{attribute addProperty ShortName ""}
FUNCTION_BLOCK ABSTRACT CUBase EXTENDS TcoCore.TcoObject IMPLEMENTS ICUBase

VAR
    _cuId        : eStations;
    _processData : ProcessDataManager(THIS^);
	_groupInspection : TcoInspectors.TcoInspectionGroup(THIS^);
	{attribute addProperty Name "<#STATUS INFO#>"}
    _statusInfo  : CUBaseStatusInfo := (Parent := THIS^);
	_operatorInfo : OperatorInfo := (Parent := THIS^);
	_settings  : CUBaseSettings := (Parent := THIS^);
	//~
	_toggle: TcoUtilities.TcoBlinker(THIS^);
	//~
	_recurringFails:CuBaseRecurringFailures:=(Parent:=THIS^);
	_productionPlaner:ProductionPlaner(THIS^);
	_internalData : REFERENCE TO InternalStorage;	
	
	{attribute clr [ReadOnly()]}
	{attribute clr [RenderIgnore()]}
	_readyForOperations : BOOL;
END_VAR

(*~
	<docu>
		<summary>
			Controls `automatic` mode of `CU00x`.
		</summary>
	</docu>
~*)
METHOD  Automat
VAR_INPUT
END_VAR
(*
	Enable condition to start `automatTask`.
	Modify according your needs.
	[! 
	THIS IS NOT SAFETY CONDITION. THE SAFETY OF PRESONNEL AND EQUIPMENT MUST BE ENSURED BY ADDITIONAL MEANS 
	TO COMPLY WITH REGULATIONS
	]
*)


AutomatTask.Task.Enabled :=  AutomatTask.Task.Busy  XOR
							(GroundTask.GroundDone AND NOT AutomatTask.Task.Busy AND THIS^.Technology.AllowAutomat(inCuId:=CuId));

(*
	Invokes `groundTask` from technology object.
*)

IF(Technology.AutomatAllTask.Execute()) THEN AutomatTask.Task.Invoke(); END_IF;

IF(Technology.ForceStepMode()) THEN
 	AutomatTask.ModeController.Mode := eSequencerMode.StepMode;
END_IF
END_METHOD

PROPERTY ABSTRACT AutomatTask : REFERENCE TO CUBaseAutomat
GET
END_GET
END_PROPERTY

PROPERTY  CreateEntityTask : TcoCore.ITcoTaskStatus
GET
CreateEntityTask := _processData._createTask;
END_GET
END_PROPERTY

PROPERTY CuId : eStations
GET
CuId := _cuId;
END_GET
SET
_cuId := CuId;
END_SET
END_PROPERTY

PROPERTY  DeleteEntityTask : TcoCore.ITcoTaskStatus
GET
DeleteEntityTask := _processData._deleteTask;
END_GET
END_PROPERTY

METHOD DoesBelong : BOOL
DoesBelong := THIS^.ProcessDataManager.Data.EntityHeader.NextStation = THIS^.CuId;
END_METHOD

METHOD EntityFlowCloseForOperations : TcoCore.ITcoTaskStatus
VAR_IN_OUT
	Header : CuHeader; 
END_VAR
THIS^.FlagCloseEntity(Header);
EntityFlowCloseForOperations := THIS^.ProcessDataManager.Update(ProcessDataManager.Data._EntityId);
END_METHOD

METHOD EntityFlowCreateNew : TcoCore.ITcoTaskStatus
VAR_INPUT
	EntityId : STRING(255);	
END_VAR
VAR_IN_OUT
	Header : CuHeader;
END_VAR
THIS^.FlagCreateNewEntity(EntityId, Header);
EntityFlowCreateNew := THIS^.ProcessDataManager.Create(EntityId);
END_METHOD

METHOD EntityFlowDiscard : TcoCore.ITcoTaskStatus
VAR_INPUT
	EntityId : STRING(255);	
END_VAR
VAR_IN_OUT	
	Header : CuHeader; 
END_VAR
THIS^.FlagThrowAwayEntity(Header);
EntityFlowDiscard := THIS^.ProcessDataManager.Update(EntityId);
END_METHOD

METHOD EntityFlowFinalize : TcoCore.ITcoTaskStatus
VAR_IN_OUT
	Header : CuHeader; 
END_VAR
THIS^.FlagFinishEntity(Header);
EntityFlowFinalize := THIS^.ProcessDataManager.Update(ProcessDataManager.Data._EntityId);
END_METHOD

METHOD EntityFlowOpenForOperations : TcoCore.ITcoTaskStatus
VAR_INPUT
	Identifier : STRING(255);	
END_VAR
VAR_IN_OUT
	Header : CuHeader;
END_VAR
EntityFlowOpenForOperations := THIS^.ProcessDataManager.Read(Identifier);
THIS^.FlagOpenEntity(Identifier, Header);
END_METHOD

PROPERTY  ExistEntityTask : TcoCore.ITcoTaskStatus
GET
ExistEntityTask := _processData._idExistsTask;
END_GET
END_PROPERTY

METHOD PRIVATE FlagCloseEntity : BOOL
VAR_IN_OUT
	Header : CuHeader; 
END_VAR
THIS^.ProcessDataManager.Data.EntityHeader.LastStation := THIS^.CuId;

IF(THIS^.ProcessDataManager.Data.EntityHeader.Results.Result = TcoInspectors.eOverallResult.Failed) THEN	
	THIS^.ProcessDataManager.Data.EntityHeader.NextStation := Header.NextOnFailed;
ELSIF(THIS^.ProcessDataManager.Data.EntityHeader.Results.Result = TcoInspectors.eOverallResult.Passed) THEN
	THIS^.ProcessDataManager.Data.EntityHeader.NextStation := Header.NextOnPassed;
ELSIF(THIS^.ProcessDataManager.Data.EntityHeader.Results.Result = TcoInspectors.eOverallResult.InProgress) THEN
	THIS^.ProcessDataManager.Data.EntityHeader.NextStation := Header.NextOnPassed;
END_IF

THIS^.ProcessDataManager.Data.EntityHeader.OpenOn := eStations.NONE;
Header.CycleTime := THIS^._statusInfo.CurrentCycleTime;
Header.CleanLoopTime := THIS^._statusInfo.CurrentCleanCycleTime;
Header.OperationsEnded := Context.RealTimeClock.NowLocal();
Header.Operator := _operatorInfo.UserName;
END_METHOD

METHOD PRIVATE FlagCreateNewEntity : BOOL
VAR_INPUT
	Identifier : STRING(255);	
END_VAR
VAR_IN_OUT
	Header : CuHeader;
END_VAR
THIS^.ProcessDataManager.Data.EntityHeader.Results.Result := TcoInspectors.eOverallResult.InProgress;
THIS^.ProcessDataManager.Data._EntityId := Identifier;
THIS^.ProcessDataManager.Data.EntityHeader.WasReset := FALSE;
END_METHOD

METHOD PRIVATE FlagFinishEntity : BOOL
VAR_IN_OUT
	Header : CuHeader; 
END_VAR
THIS^.ProcessDataManager.Data.EntityHeader.LastStation := THIS^.CuId;

IF(THIS^.ProcessDataManager.Data.EntityHeader.Results.Result = TcoInspectors.eOverallResult.InProgress) THEN
	THIS^.ProcessDataManager.Data.EntityHeader.Results.Result := TcoInspectors.eOverallResult.Passed;
END_IF

IF(THIS^.ProcessDataManager.Data.EntityHeader.Results.Result = TcoInspectors.eOverallResult.Failed) THEN	
	THIS^.ProcessDataManager.Data.EntityHeader.NextStation := Header.NextOnFailed;
ELSIF(THIS^.ProcessDataManager.Data.EntityHeader.Results.Result = TcoInspectors.eOverallResult.Passed) THEN
	THIS^.ProcessDataManager.Data.EntityHeader.NextStation := Header.NextOnPassed;
END_IF

THIS^.ProcessDataManager.Data.EntityHeader.OpenOn := eStations.NONE;

Header.CycleTime := THIS^._statusInfo.CurrentCycleTime;
Header.CleanLoopTime := THIS^._statusInfo.CurrentCleanCycleTime;
Header.OperationsEnded := Context.RealTimeClock.NowLocal();
Header.Operator := _operatorInfo.UserName;
END_METHOD

METHOD PRIVATE FlagOpenEntity : BOOL
VAR_INPUT
	Identifier : STRING(255);	
END_VAR
VAR_IN_OUT
	Header : CuHeader;
END_VAR
Header.Operator := _operatorInfo.UserName;
Header.OperationsStarted := Context.RealTimeClock.NowLocal();
THIS^.ProcessDataManager.Data.EntityHeader.Results.Result := TcoInspectors.eOverallResult.InProgress;
THIS^.ProcessDataManager.Data._EntityId := Identifier;
THIS^.ProcessDataManager.Data.EntityHeader.OpenOn := THIS^.CuId;
THIS^.ProcessDataManager.Data.EntityHeader.WasReset := FALSE;
END_METHOD

METHOD PRIVATE FlagThrowAwayEntity : BOOL
VAR_IN_OUT	
	CuHeader : CuHeader; 
END_VAR
IF(THIS^.ProcessDataManager.Data.EntityHeader.OpenOn <> eStations.NONE) THEN
	THIS^.ProcessDataManager.Data.EntityHeader.LastStation := THIS^.CuId;
	THIS^.ProcessDataManager.Data.EntityHeader.NextStation := CuHeader.NextOnFailed;
	THIS^.ProcessDataManager.Data.EntityHeader.Results.Result := TcoInspectors.eOverallResult.Failed;
	THIS^.ProcessDataManager.Data.EntityHeader.WasReset := TRUE;
END_IF;
END_METHOD

(*~
	<docu>
		<summary>
			Controls `ground` mode of `CU00x`.
		</summary>
	</docu>
~*)
METHOD Ground : BOOL
VAR_INPUT
END_VAR
(*
	Enable condition to start `groundTask`.
	Modify according your needs.
	[! 
	THIS IS NOT SAFETY CONDITION. THE SAFETY OF PRESONNEL AND EQUIPMENT MUST BE ENSURED BY ADDITIONAL MEANS 
	TO COMPLY WITH REGULATIONS
	]
*)

GroundTask.Task.Enabled :=  THIS^.Technology.AllowGround(inCuId:=CuId)  OR GroundTask.Task.Busy ;

(*
	Invokes `groundTask` from technology object.
*)


IF(Technology.GroundAllTask.Execute()) THEN GroundTask.Restore();GroundTask.Task.Invoke(); END_IF;


IF GroundTask.GroundDone AND GroundTask.Task.Execute() THEN GroundTask.Restore();GroundTask.Task.Invoke();END_IF;
END_METHOD

PROPERTY ABSTRACT GroundTask : REFERENCE TO CUBaseGround
GET
END_GET
END_PROPERTY

PROPERTY FINAL GroupInspection : REFERENCE TO TcoInspectionGroup
GET
GroupInspection REF= _groupInspection;
END_GET
END_PROPERTY

(*~
	<docu>
		<summary>
			Code to be called cylically when `CU00x` idle; no other mode is active.
		</summary>
	</docu>
~*)
METHOD Idle : BOOL
END_METHOD

METHOD InternalCloseEntity : BOOL
VAR_INPUT
	inCarrier : UINT;
	refStorage : REFERENCE TO InternalStorage;
END_VAR
VAR_IN_OUT
	inoHeader : CuHeader; 
END_VAR
VAR_INST
	_internalData : REFERENCE TO InternalStorage;	
END_VAR
THIS^.FlagCloseEntity(inoHeader);
_internalData REF= refStorage;
InternalCloseEntity := _internalData.SaveByCarrier(inCarrier, THIS^.ProcessDataManager.Data);
END_METHOD

METHOD InternalCreateNewEntity : BOOL
VAR_INPUT
	inCarrier : UINT;
	refStorage : REFERENCE TO InternalStorage;
END_VAR
VAR_IN_OUT
	inoHeader : CuHeader; 
END_VAR
VAR_INST
	_internalData : REFERENCE TO InternalStorage;	
END_VAR
THIS^.FlagCreateNewEntity(UINT_TO_STRING(inCarrier), inoHeader);
THIS^.ProcessDataManager.Data.EntityHeader.Carrier := UINT_TO_STRING(inCarrier);
_internalData REF= refStorage;
InternalCreateNewEntity := _internalData.SaveByCarrier(inCarrier, THIS^.ProcessDataManager.Data);
END_METHOD

METHOD InternalFinishEntity : BOOL
VAR_INPUT
	inCarrier : UINT;
	refStorage : REFERENCE TO InternalStorage;
END_VAR
VAR_IN_OUT
	inoHeader : CuHeader; 
END_VAR
VAR_INST
	_internalData : REFERENCE TO InternalStorage;	
END_VAR
THIS^.FlagFinishEntity(inoHeader);

_internalData REF= refStorage;
InternalFinishEntity := _internalData.SaveByCarrier(inCarrier, THIS^.ProcessDataManager.Data);
END_METHOD

METHOD InternalOpenEntity : BOOL
VAR_INPUT
	inCarrier : UINT;
	refStorage : REFERENCE TO InternalStorage;
END_VAR
VAR_IN_OUT
	inoHeader : CuHeader; 
END_VAR
VAR_INST
	_internalData : REFERENCE TO InternalStorage;	
END_VAR
_internalData REF= refStorage;
InternalOpenEntity := _internalData.GetByCarrier(inCarrier, THIS^.ProcessDataManager.Data);
THIS^.FlagOpenEntity(UINT_TO_STRING(inCarrier), inoHeader);
END_METHOD

METHOD InternalRetrieveEntity : BOOL
VAR_INPUT
	inCarrier : UINT;
	refStorage : REFERENCE TO InternalStorage;
END_VAR
VAR_INST
	_internalData : REFERENCE TO InternalStorage;	
END_VAR
_internalData REF= refStorage;
InternalRetrieveEntity := _internalData.GetByCarrier(inCarrier, THIS^.ProcessDataManager.Data);
END_METHOD

METHOD InternalThrowAwayEntity : BOOL
VAR_INPUT
	inCarrier : UINT;
	refStorage : REFERENCE TO InternalStorage;
END_VAR
VAR_IN_OUT
	inoHeader : CuHeader; 
END_VAR
VAR_INST
	_internalData : REFERENCE TO InternalStorage;	
END_VAR
THIS^.FlagThrowAwayEntity(inoHeader);
_internalData REF= refStorage;
InternalThrowAwayEntity := _internalData.SaveByCarrier(inCarrier, THIS^.ProcessDataManager.Data);
END_METHOD

(*~
	<docu>
		<summary>
			Controls `manual` mode of `CU00x`.
		</summary>
	</docu>
~*)
METHOD Manual : BOOL
VAR_INPUT
END_VAR
(*
	Enable condition to start `automatTask`.
	Modify according your needs.
	[! 
	THIS IS NOT SAFETY CONDITION. THE SAFETY OF PRESONNEL AND EQUIPMENT MUST BE ENSURED BY ADDITIONAL MEANS 
	TO COMPLY WITH REGULATIONS
	]
*)

ManualTask.Task.Enabled :=  THIS^.Technology.AllowManual(inCuId:=CuId)  OR ManualTask.Task.Busy;
END_METHOD

PROPERTY ABSTRACT ManualTask : REFERENCE TO TcoTaskedService
GET
END_GET
END_PROPERTY

PROPERTY FINAL ProcessDataManager : REFERENCE TO ProcessDataManager
GET
ProcessDataManager REF= _processData;
END_GET
END_PROPERTY

PROPERTY  ReadEntityTask : TcoCore.ITcoTaskStatus
GET
ReadEntityTask := _processData._readTask;
END_GET
END_PROPERTY

METHOD ReadyForOperations : BOOL
VAR_INPUT
END_VAR
ReadyForOperations := _readyForOperations;
END_METHOD

PROPERTY ABSTRACT RecoverTask : REFERENCE TO CUBaseRecover
GET
END_GET
END_PROPERTY

PROPERTY RecurringFails : REFERENCE TO CuBaseRecurringFailures
GET
RecurringFails REF= _recurringFails;
END_GET
END_PROPERTY

METHOD ResetReadyForOperations : BOOL
_readyForOperations := false;
END_METHOD

METHOD  RunOperations : BOOL
VAR_INPUT
	refGlobalTrigger:REFERENCE TO BOOL;
END_VAR
VAR
	_trrigger:REFERENCE TO BOOL;
END_VAR
_trrigger REF=refGlobalTrigger;
RunOperations := _trrigger;
END_METHOD

METHOD  SetReadyForOperations : BOOL
VAR_INPUT
END_VAR
_readyForOperations := TRUE;
END_METHOD

PROPERTY ABSTRACT StatusInfo : REFERENCE TO CUBaseStatusInfo
GET
END_GET
END_PROPERTY

PROPERTY ABSTRACT SuspendTask : REFERENCE TO CUBaseSuspend
GET
END_GET
END_PROPERTY

PROPERTY Technology : REFERENCE TO Technology
GET
VAR
    _technology : POINTER TO Technology;
END_VAR
IF __QUERYPOINTER(Parent, _technology) THEN // Check if _Parent is Station001
    Technology REF= _technology^;              // If the check is successful dereference a pointer. simlar to THIS^ or SUPER^
END_IF
END_GET
END_PROPERTY

PROPERTY PUBLIC ToggleBlinker : REFERENCE TO TcoUtilities.TcoBlinker
GET
ToggleBlinker ref= _toggle;
END_GET
END_PROPERTY

PROPERTY  UpdateEntityTask : TcoCore.ITcoTaskStatus
GET
UpdateEntityTask := _processData._updateTask;
END_GET
END_PROPERTY

METHOD UpdateInfo : BOOL
VAR_INPUT
END_VAR
_toggle(inOffTime:=T#500MS,inOnTime:=T#500MS);

IF AutomatTask.ClearCounterDataTask.Execute() THEN
	AutomatTask.ClearCounter();
	AutomatTask.ClearCounterDataTask.DoneWhen(TRUE);
END_IF

_statusInfo.State := eCUState.None;

IF _statusInfo.CurrentCleanCycleTime  >= _settings.WarningCycleTime
	AND _statusInfo.CurrentCleanCycleTime  < _settings.ErrorCycleTime THEN
	_statusInfo.State:= eCUState.HasWarning;
ELSIF _statusInfo.CurrentCleanCycleTime   >= _settings.ErrorCycleTime THEN
	_statusInfo.State := eCUState.HasError;
END_IF; 


IF _toggle.IsOff THEN
	_statusInfo.State := eCUState.None;
END_IF



IF AutomatTask.Task.Busy THEN

    _statusInfo.Mode                   := eCUMode.AutomatMode;
    _statusInfo.CurrentTaskDescription := '<#AUTOMAT#>';
    _statusInfo.CurrentCycleTime       := AutomatTask._SequenceElapsedTime;
	_statusInfo.CurrentCleanCycleTime  := T#0S;

	IF AutomatTask._startCleanCycleTime<>T#0S AND AutomatTask._stopCleanCycleTime=T#0S  THEN
		_statusInfo.CurrentCleanCycleTime  := AutomatTask._SequenceElapsedTime-AutomatTask._startCleanCycleTime;
	ELSIF AutomatTask._stopCleanCycleTime<>T#0S  THEN
		_statusInfo.CurrentCleanCycleTime  := AutomatTask._stopCleanCycleTime-AutomatTask._startCleanCycleTime;
	ELSE
		_statusInfo.CurrentCleanCycleTime :=AutomatTask._startCleanCycleTime;
	END_IF;
	
	_statusInfo.AverageCycleTime	   := AutomatTask.AverageCycleTime;
	_statusInfo.AverageCleanCycleTime  := AutomatTask.AverageCleanCycleTime;
    _statusInfo.CurrentUid             := AutomatTask.CurrentStep.ID;
    _statusInfo.CurrentOperation       := AutomatTask.CurrentStep.Description;
    _statusInfo.CurrentIsInStepMode    := AutomatTask._modeController._mode = eSequencerMode.StepMode;
ELSIF GroundTask.Task.Busy THEN
    _statusInfo.Mode := eCUMode.GroundMode;
	_statusInfo.CurrentTaskDescription := '<#GROUND#>';
    _statusInfo.CurrentCycleTime       := GroundTask._SequenceElapsedTime;
	_statusInfo.CurrentCleanCycleTime := T#0S;
	_statusInfo.AverageCycleTime	   := GroundTask.AverageCycleTime;
	_statusInfo.AverageCleanCycleTime  := T#0S;
    _statusInfo.CurrentUid             := GroundTask.CurrentStep.ID;
    _statusInfo.CurrentOperation       := GroundTask.CurrentStep.Description;
    _statusInfo.CurrentIsInStepMode    := GroundTask._modeController._mode = eSequencerMode.StepMode;
ELSIF THIS^.ManualTask.Busy THEN
    _statusInfo.Mode := eCUMode.ManualMode;
	_statusInfo.CurrentTaskDescription := '<#MANUAL#>';
	_statusInfo.State := eCUState.None;
	_statusInfo.CurrentIsInStepMode    := FALSE;

ELSIF THIS^.GroundTask.Task.Done THEN
	_statusInfo.CurrentTaskDescription := '<#READY TO START#>';
	_statusInfo.Mode := eCUMode.GroundModeDone;
	_statusInfo.CurrentCycleTime       := GroundTask._SequenceElapsedTime;
    _statusInfo.CurrentUid             := GroundTask.CurrentStep.ID;
    _statusInfo.CurrentOperation       := GroundTask.CurrentStep.Description;
    _statusInfo.CurrentIsInStepMode    := GroundTask._modeController._mode = eSequencerMode.StepMode;
	_statusInfo.State := eCUState.None;

ELSE
    _statusInfo.Mode := eCUMode.NoMode;	
	_statusInfo.CurrentTaskDescription := '<#IDLE#>';
	_statusInfo.CurrentCycleTime       := T#0S;
    _statusInfo.CurrentUid             := 0;
    _statusInfo.CurrentOperation       := '';
    _statusInfo.CurrentIsInStepMode    := FALSE;
	_statusInfo.State := eCUState.None;
END_IF
END_METHOD

END_FUNCTION_BLOCK

(* stored: Version 1.1.0.1
   POU CUBase: Id {7de2193c-318e-4c64-a9a6-ba23fb2e4da1}, SpecialFunc None
   Folder Misc: Id {89a011fb-946c-4af2-b16f-4abd86442495}
   Folder Modes: Id {d650a7bf-6367-4a6c-a191-a985e54df897}
   Folder ProcessData: Id {1a8aa84b-31e4-41aa-b103-fbb20e0c7128}
   Folder CrudTaskState: Id {3cbcef83-2f8f-092f-1642-2d5bb3f25f3f}
   Folder DataFlaging: Id {aed3d7b3-4fd1-0c13-2eed-417fc6b5b252}
   Folder ExternalData: Id {8389998d-539c-07b7-2bed-035331c1a0d8}
   Folder InternalData: Id {5ea75a1d-a09d-4e05-8586-dc704b6c3cc3}
   Folder RecurringFailures: Id {aea7587e-0f13-0992-2127-c34de6e860fe}
   Folder Tasks: Id {522e67de-7340-4416-b0c7-f54a63e10aed}
   Method Automat: Id {a2102426-ef76-401d-8346-4b915f2c9694}
   Property AutomatTask: Id {9a1989f3-7511-4b12-80ce-78bb1add06c6}
   Get Get: Id {86426d31-47b7-4512-bf28-f740d21d447d}
   Property CreateEntityTask: Id {8d9f994a-39cb-072a-20b7-6e45f0e751c3}
   Get Get: Id {25505615-9457-08c9-0598-a426211f4721}
   Property CuId: Id {65aa5bdf-9849-470a-831e-c3ba5e79392e}
   Get Get: Id {c66b2e7b-b895-4144-891c-99fd374ac89f}
   Set Set: Id {07920021-9ea4-4f22-9984-168c54ee5866}
   Property DeleteEntityTask: Id {904e79cf-1b7d-0b16-004d-f7a93864b5a8}
   Get Get: Id {3aaafc1d-63ff-0db7-27cf-f78743af539c}
   Method DoesBelong: Id {55fc80ad-32c7-442e-a227-eb2402c499aa}
   Method EntityFlowCloseForOperations: Id {8bf49847-55ad-09e2-18b7-e269b9aac41c}
   Method EntityFlowCreateNew: Id {def96a3d-be60-022c-22e1-cec3782e9b03}
   Method EntityFlowDiscard: Id {e706bdf6-bfe5-0d86-0aa7-1e9e631ad7f3}
   Method EntityFlowFinalize: Id {d334eb15-8a45-08f2-3686-ad4133f632f2}
   Method EntityFlowOpenForOperations: Id {9ce16e44-9451-0ab8-22fc-14904cbb8438}
   Property ExistEntityTask: Id {97b85c56-ca7a-0f33-3276-6bd0c596f8b5}
   Get Get: Id {0af78185-edfb-0a12-0373-dc5b82f7228b}
   Method FlagCloseEntity: Id {f071be0b-9fd5-042e-3314-968c40af4466}
   Method FlagCreateNewEntity: Id {f5c3e5fb-7bd4-04c3-3dc2-2885f9b6d068}
   Method FlagFinishEntity: Id {a410cec9-47a6-0ae5-021f-0adac5adedb9}
   Method FlagOpenEntity: Id {f1aa0c9c-4f3a-0a38-0281-19b168846e2a}
   Method FlagThrowAwayEntity: Id {ab780eac-b9e9-0133-03b0-8c9a606ed51c}
   Method Ground: Id {6ef710e9-01db-4ecc-94fc-dcc146d80f72}
   Property GroundTask: Id {6cf29f50-dec8-49c6-a97a-8a93927ca757}
   Get Get: Id {41f5a2de-fade-47b5-8a6c-d888d0eac9c5}
   Property GroupInspection: Id {e13fb714-68d8-429d-a303-f7e6cff57930}
   Get Get: Id {3baebd85-3b43-4308-98fa-016c2bb452b8}
   Method Idle: Id {e87c0f97-9703-4da3-9774-ed86bd6184b7}
   Method InternalCloseEntity: Id {dfea0e83-d826-46d9-999d-a40573b91b00}
   Method InternalCreateNewEntity: Id {2a260e96-2965-4d92-91e5-527d8ec911bc}
   Method InternalFinishEntity: Id {f4f6b5d3-650a-43ef-93bf-662dc33f326f}
   Method InternalOpenEntity: Id {c2a47fa2-fa48-4474-91bc-486ebcf5d6f6}
   Method InternalRetrieveEntity: Id {4e223708-c43d-4037-a2dd-eac052151e43}
   Method InternalThrowAwayEntity: Id {e3889063-3943-4256-b512-d2920a6f746b}
   Method Manual: Id {ca59dfc2-4891-4382-ac63-95609aefa41f}
   Property ManualTask: Id {a2025997-47b5-45e1-80f0-0c1e8cce860d}
   Get Get: Id {c93ae827-0df1-40b0-b0fa-7bfc00959641}
   Property ProcessDataManager: Id {95e82431-3124-4f70-be63-551f0ca81c55}
   Get Get: Id {75873f97-0e26-4094-bf28-402fb0488241}
   Property ReadEntityTask: Id {e052507d-c99d-0b49-2b30-e3a644be24d4}
   Get Get: Id {77518d1e-59e8-0173-1e59-63b515f69430}
   Method ReadyForOperations: Id {77a708be-476c-4f16-9146-a2c225c4a4d4}
   Property RecoverTask: Id {3e03c8f5-0e6a-4257-b8ec-f05883753522}
   Get Get: Id {b652b901-2fff-46c7-8e8d-0292570c5ddc}
   Property RecurringFails: Id {c6ba4858-160c-006e-34fa-84af07e0038f}
   Get Get: Id {95d834e8-2609-0f13-155a-8ef6c95bef05}
   Method ResetReadyForOperations: Id {8bdd63cb-1ddc-4a3a-8a46-b497c45dd233}
   Method RunOperations: Id {a957592c-a5b8-4fd8-8056-4beaed2d9ff5}
   Method SetReadyForOperations: Id {58953506-ec17-4f2c-a7ed-ed0c9eabd4ea}
   Property StatusInfo: Id {8869b0c0-1b6b-4ea5-bfe7-ba8752959d51}
   Get Get: Id {6df77d60-346a-4f90-8a89-5b3120d43b1f}
   Property SuspendTask: Id {304bee79-70a6-4794-aa3f-17793994512b}
   Get Get: Id {a51ffe0f-2bc2-47f1-94e4-a1c50b8b115a}
   Property Technology: Id {9acc4c59-d4d2-4ccd-a7ca-7b094f3f86e5}
   Get Get: Id {a26286e4-0ce6-43b9-8eee-d2e9be8bc503}
   Property ToggleBlinker: Id {0ed49b78-0603-4128-ab5c-75f37242700d}
   Get Get: Id {283c9d38-3bff-4a7f-abd0-6cf25f97bb1d}
   Property UpdateEntityTask: Id {05c804c9-7f4b-0e37-2ebf-2fe6f3b9eb66}
   Get Get: Id {efded1af-2b8a-0cbf-039b-3695e9082143}
   Method UpdateInfo: Id {d2563fa9-29cd-48cb-9533-a53a49a45068} *)
